TYPE CoverIOStatuses :
STRUCT
	///Is the I/O in a healthy state?
	healthStatus: HealthStatus;
END_STRUCT
END_TYPE

(* stored: Version 1.1.0.1, ProductVersion 3.1.4019.2
   DUT CoverIOStatuses: Id {de4ff81c-2292-41ef-a138-7a0658f656ab} *)
